// TIA Portal V18 export
FUNCTION "Funktion1" : Void   // FC1, FBD
{ S7_Optimized_Access := 'TRUE' }
VERSION : 0.1
// stored: AutoNumber true, IsIECCheckEnabled false, SetENOAutomatically false, UDAEnableTagReadback false
   VAR_INPUT
      Input : Bool;
   END_VAR
   VAR_OUTPUT
      Output_1 : Bool;
   END_VAR
BEGIN
END_FUNCTION
